TYPE ST_TcMatSimObjectDataAreaInfo_1 :
STRUCT
	pPlcVar: PVOID;
	pModuleProcImg: PVOID;
	nSize: UDINT;
	nDataAreaId: UDINT;
	eDataAreaType: E_TcMatSimDataAreaType;
END_STRUCT
END_TYPE

(* stored: Version 1.1.0.1, ProductVersion 3.1.4020.12
   DUT ST_TcMatSimObjectDataAreaInfo_1: Id {16297a9c-7688-4514-b16b-d328ad0fd721} *)
